{attribute 'linkalways'} 
{attribute 'no_explicit_call' := 'This FB is a CLASS and must be accessed using methods or properties'}
{attribute 'enable_dynamic_creation'}
FUNCTION_BLOCK MockNumericDatatype_INT EXTENDS NumericDatatypeBase
VAR
	localData : INT;
	activeData : REFERENCE TO INT REF= localData;
END_VAR

PROPERTY PUBLIC Address : PVOID
GET
Address := ADR(activeData);
END_GET
END_PROPERTY

METHOD PUBLIC ClearReference
VAR_INPUT
END_VAR
activeData REF= localData;
END_METHOD

METHOD PUBLIC Clone : I_Datatype
VAR
    pClone : POINTER TO MockNumericDatatype_INT;
END_VAR
pClone := __NEW(MockNumericDatatype_INT(InitialValue := Value));
Clone := pClone^;
END_METHOD

METHOD FB_init : BOOL
VAR_INPUT
	bInitRetains : BOOL; // if TRUE, the retain variables are initialized (warm start / cold start)
	bInCopyCode : BOOL;  // if TRUE, the instance afterwards gets moved into the copy code (online change)
	InitialValue : INT;
END_VAR
localData := InitialValue;
END_METHOD

PROPERTY PUBLIC IsFloat : BOOL
GET
IsFloat := FALSE;
END_GET
END_PROPERTY

PROPERTY PUBLIC IsSigned : BOOL
GET
IsSigned := TRUE;
END_GET
END_PROPERTY

METHOD PUBLIC MakeReferenceTo
VAR_INPUT
	ReferenceTarget : REFERENCE TO INT;
END_VAR
activeData REF= ReferenceTarget;
END_METHOD

PROPERTY PUBLIC MaxValue : INT
GET
MaxValue := DatatypeLimits.INT_MAX_VALUE;
END_GET
END_PROPERTY

PROPERTY PUBLIC MinValue : INT
GET
MinValue := DatatypeLimits.INT_MIN_VALUE;
END_GET
END_PROPERTY

METHOD PROTECTED SerializeMaxValue
VAR_INPUT
	Serializer : I_Serializer;
END_VAR
Serializer.AddInt(MaxValue);
END_METHOD

METHOD PROTECTED SerializeMinValue
VAR_INPUT
	Serializer : I_Serializer;
END_VAR
Serializer.AddInt(MinValue);
END_METHOD

METHOD PUBLIC SerializeWith
VAR_INPUT
	Serializer : I_Serializer;
END_VAR
Serializer.AddInt(activeData);
END_METHOD

PROPERTY PUBLIC Size : UDINT
GET
Size := SIZEOF(activeData);
END_GET
END_PROPERTY

METHOD TryDeserializeFrom : BOOL
VAR_INPUT
	Deserializer : I_Deserializer;
	Feedback : I_DeserializerFeedback;
END_VAR
TryDeserializeFrom := Deserializer.TryGetInt(activeData, Feedback);
END_METHOD

METHOD TryMakeReferenceTo : BOOL
VAR_INPUT
	Target : I_Datatype;
END_VAR
VAR
	pTargetData : POINTER TO INT;
END_VAR
IF NOT (Target.TypeName = TypeName) THEN
	RETURN;
END_IF

pTargetData := Target.Address;
activeData REF= pTargetData^;
TryMakeReferenceTo := TRUE;
END_METHOD

PROPERTY PUBLIC TypeName : T_MAXSTRING
GET
TypeName := 'INT';
END_GET
END_PROPERTY

PROPERTY PUBLIC Value : REFERENCE TO INT
GET
Value REF= activeData;
END_GET
END_PROPERTY

END_FUNCTION_BLOCK

(* stored: Version 1.1.0.1, ProductVersion 3.1.4024.12
   POU MockNumericDatatype_INT: Id {9a96c563-0c5f-4762-a707-bd3f7b261a4c}, SpecialFunc None
   Folder Constructor: Id {08e10cec-c835-4150-a7c9-ae41abead9f4}
   Folder Protected: Id {56b22893-8e97-444b-a694-a00cb5e06d58}
   Property Address: Id {98257829-3f0b-4260-af53-f3549dacae22}
   Get Get: Id {f6f62f84-56ba-4bc4-ab3b-6cb699cb4057}
   Method ClearReference: Id {1f529931-3f49-4d36-8bb6-26739a21766f}
   Method Clone: Id {46eb6cc3-7af6-4f01-8396-1a38f47b2886}
   Method FB_init: Id {7add3e91-7cf2-4a24-bd54-f6b2ee4a69d8}
   Property IsFloat: Id {5d18eb5a-06eb-4c6d-ad82-b5375f671115}
   Get Get: Id {663f6e1a-42db-43ef-8497-664b52c0e104}
   Property IsSigned: Id {087b14db-2532-448a-a906-f49537e546d1}
   Get Get: Id {539a6319-d371-4611-bfb7-56788d86a75a}
   Method MakeReferenceTo: Id {576fb395-a119-4204-bd1a-bd8fabdca254}
   Property MaxValue: Id {13bf50c2-95ee-4f97-a110-dd0955ea1a6e}
   Get Get: Id {845f3f35-29c0-429a-96b4-fbae8b8b4fb8}
   Property MinValue: Id {80021b87-783d-4c60-bb0f-cdf9e0ca4cba}
   Get Get: Id {e9503079-778a-4ed5-ae8f-acc1d453b00c}
   Method SerializeMaxValue: Id {094b3350-c4a4-429d-80de-082ed9fda8b9}
   Method SerializeMinValue: Id {48a3cbe3-ade6-44cb-a1f8-e7a9f9b21508}
   Method SerializeWith: Id {e328b6c6-dc72-410f-8e3b-68e369940afa}
   Property Size: Id {349094fb-fadc-4e18-bced-0668a7b07409}
   Get Get: Id {64421bcd-ec3e-4b32-af1d-a522d55eea61}
   Method TryDeserializeFrom: Id {b5fd1959-a56e-4b2a-b390-e63ef56f4338}
   Method TryMakeReferenceTo: Id {132eda61-bf72-4f75-bd92-572d04312011}
   Property TypeName: Id {518e6cdc-db74-46e8-8860-922105556ac6}
   Get Get: Id {6bc09f9f-5b95-4e80-8c1d-89f7003f7d90}
   Property Value: Id {fd3f6fff-e182-4b74-98c8-3d62616219fe}
   Get Get: Id {096e268a-dd35-4b90-9ca7-50b3877daf0f} *)
